{attribute 'GeneratedUsingTerminal: EL6001-0000-0020'}
{attribute addProperty BoxType "EL6001-0000-0020"}
{attribute addProperty Id "StatusAT %I*UINT2Data_InAT %I*ARRAY[0..21] OF USINT22"}
{attribute addProperty CRC "1367962124"}
{attribute addProperty Size "24"}
TYPE Inputs_6C2FC202 EXTENDS InputBase_8311D824 :
STRUCT
	{attribute addProperty Name "Status"}
	Status AT %I* : UINT;
	{attribute addProperty Name "Data_In"}
	Data_In AT %I* : ARRAY[0..21] OF USINT;
END_STRUCT
END_TYPE

(* stored: Version 1.2.0.0, ProductVersion 3.1.4024.9
   DUT Inputs_6C2FC202: Id {35245bce-20bb-4450-8f55-5418df574737} *)
